// TwinCAT 3 PLC project Untitled1
// ProgramVersion: 3.1.4024.0
// libraries:
//   Tc2_Standard, * (Beckhoff Automation GmbH)
//   Tc2_System, * (Beckhoff Automation GmbH)
//   Tc3_Module, * (Beckhoff Automation GmbH)
// project tree:
//   GVLs/ GVL.TcGVL
//   POUs/ GetWaterDuration.TcPOU, MonitoringTheSoilTask.TcPOU, WateringTask.TcPOU
// real-time tasks:
//   TASK PlcTask: cycle T#10ms, priority 20, ADS port 350

// ---- GVLs/GVL.TcGVL
{attribute 'qualified_only'}
VAR_GLOBAL
Moisture : REAL :=50; // Represent the soil moisture
Temp : REAL := 25; // Shows the temperature in Celsius
WaterRequired : BOOL := FALSE; // Tells if water is needed
WaterON : BOOL := FALSE; // Pump is on
WaterDuration : TIME :=T#0S;// Tell watering period
END_VAR

// ---- POUs/GetWaterDuration.TcPOU
FUNCTION GetWaterDuration : TIME
VAR_INPUT
	MoistIn:REAL ;
	TempIn:REAL;
END_VAR

GetWaterDuration:= REAL_TO_TIME(10 + (TempIn - 20) - (MoistIn * 0.1)) * T#1S;
IF GetWaterDuration < T#5S THEN GetWaterDuration :=T#5S; END_IF;
IF GetWaterDuration > T#20S THEN GetWaterDuration :=T#20S; END_IF;

END_FUNCTION

// ---- POUs/MonitoringTheSoilTask.TcPOU
PROGRAM MonitoringTheSoilTask
VAR
	Timer: TON;
	state: INT;
	Moisture: REAL;
	Temp: REAL;
	WaterRequired: BOOL;
END_VAR

0

CASE state OF
	0:// Initial position
	Moisture :=50;
	Temp := 25;
	state :=1;
	
	1: //ReadSensors
	Moisture:= Moisture - 1
	IF Moisture < 0 THEN Moisture :=0 END_IF;
	Temp := Temp;
	state := 2;
	 
	2://UpdateGVL
	WaterRequired := (Moisture <30 AND Temp > 20 );
	State:=1;

	
	
	
	
END_CASE

END_PROGRAM

// ---- POUs/WateringTask.TcPOU
PROGRAM WateringTask
VAR
	WaterTimer: TON;
state : INT	 :=0; 	
Delay: Ton;
END_VAR

 	
//Watering control
CASE state OF
	
END_CASE
0:// Initial position
WaterON:= FALSE;
state:=1;
1:// Checking the conditions
IF WaterRequired THEN
            WaterDuration := GetWaterDuration(Moisture, Temp);
            WaterOn := TRUE;
            WaterTimer(IN := TRUE, PT := WaterDuration);
            nState := 2;
        ELSE
            nState := 3;
        END_IF;
		
2:  // Watering
WaterTimer(IN := TRUE);
        IF WaterTimer.Q THEN
          WaterON := FALSE;
WaterRequired := FALSE;
WaterTimer(IN := FALSE);
            state := 3;
3:// Idle
Delay(IN:=TRUE, PT:=T#5S);
IF NOT(Delay.Q) THEN
	RETURN;
END_IF
Delay(In:=FALSE);
state:=1;		
END_CASE

END_PROGRAM
